PROGRAM Shutdown
VAR
	bStart	AT%I* : BOOL := FALSE;
	Shutdown_Block: NT_Shutdown;
END_VAR

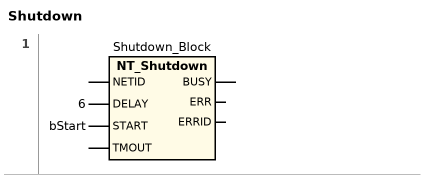
// NETWORK 1
Shutdown_Block(DELAY := 6, START := bStart); // NT_Shutdown

END_PROGRAM

(* stored: Version 1.1.0.1, ProductVersion 3.1.4022.3
   POU Shutdown: Id {073131ec-e0ca-411a-8578-ca755403f180}, SpecialFunc None *)
